(* CODESYS project SM_RTD.library
   Description: Device support for RTD Data Acquisition 8-Layer Stackable HAT for Raspberry Pi
   Version: 1.1.0.0
   Title: Raspberry I2C RTD Data Acquisition
   Author: Sequent Microsystems
   DocFormat: reStructuredText
   Placeholder: PlaceholderTemplate
   LanguageModelAttribute: qualified-access-only
   Company: Sequent Microsystems
   DefaultNamespace: SM_RTD

Project tree, tasks and I/O mapping:
  libraries: Raspberry Pi Peripherals, 4.6.0.0 (3S - Smart Software Solutions GmbH); IoStandard, 3.5.17.0 (System); Standard, 3.5.18.0 (System)
  global variables GVL
  function block SM_RTD [ST]: AfterReadInputs, BeforeWriteOutputs
  Library Information/
    function GetLibVersionNumber [ST]
    function GetLibVersion [ST]
    function IsLibReleased [ST]
  Project Information/
    function GetCompany [ST]
    function GetTitle [ST]
    function GetVersion [ST]
    function GetTextProperty [ST]
    function GetTextProperty2 [ST]
    function GetNumberProperty [ST]
    function GetBooleanProperty [ST]
    function GetVersionProperty [ST]
  data type REAL_UNION
*)

// REAL_UNION
TYPE REAL_UNION :
UNION
	rVal: REAL;
	b : ARRAY[0..3] OF BYTE;
END_UNION
END_TYPE

// GVL
//{attribute 'qualified_only'}
VAR_GLOBAL CONSTANT
	RTD_VAL_ADD: USINT := 16#00;	
END_VAR

// SM_RTD
FUNCTION_BLOCK SM_RTD EXTENDS i2c
VAR_INPUT
	//relayState: ARRAY[0..7] OF BOOL;
END_VAR
VAR_OUTPUT
	inRtdTemp: ARRAY[0..7] OF REAL;
END_VAR
VAR
	timer: TON := (IN:=TRUE);
END_VAR
VAR_TEMP	
	i, usi: USINT;
	buff: ARRAY[0..20] OF USINT;	
END_VAR

SUPER^();

CASE _iState OF
0:
	IF usiAddress < 16#40 OR  usiAddress > 16#47 THEN
		usiAddress := 16#40;
	END_IF
	
	IF SUPER^.init() THEN
		_iState := 5;
	END_IF	
5:	
	Timer.pt := T#25MS;
	
	// no initialisation here
	
	
	_iState := 10;
END_CASE

METHOD AfterReadInputs:INT
VAR
	Buffer : ARRAY[0..3] OF BYTE;
	ch: USINT;
	address: USINT;
	value: REAL_UNION;
	len: DINT;	
END_VAR
SUPER^.AfterReadInputs();

IF _iState = 10 THEN
	timer(IN:=TRUE);
	IF timer.Q THEN	
		FOR ch:=0 TO 7 DO
			address:= RTD_VAL_ADD + 4*ch;
			len := readregister(address, ADR(Buffer), 4);		
			IF len = 4 THEN
				value.b := Buffer;
				inRtdTemp[ch] := value.rVal;
				
			END_IF
		END_FOR
		
		timer(IN:=FALSE);
	END_IF
END_IF
END_METHOD

METHOD BeforeWriteOutputs:INT
VAR
	i: USINT;
	cnt: USINT;
	inVal:UINT;
	inSVal:USINT;
	buff: ARRAY[0..2] OF USINT;
	wStat: BOOL;
END_VAR
SUPER^.BeforeWriteOutputs();

IF _iState = 10 THEN

//nothing to write			
END_IF
END_METHOD

END_FUNCTION_BLOCK

// Library Information/GetLibVersionNumber
// This function has been automatically generated from the project information.
FUNCTION GetLibVersionNumber : DWORD
VAR_INPUT
	
END_VAR

GetLibVersionNumber := 16842752;

END_FUNCTION

// Project Information/GetCompany
// This function has been automatically generated from the project information.
{attribute 'signature_flag' := '1073741824'}
{attribute 'register_in_runtime'}
FUNCTION GetCompany : WSTRING
VAR_INPUT
	
END_VAR

GetCompany := "Sequent Microsystems";

END_FUNCTION

// Project Information/GetTitle
// This function has been automatically generated from the project information.
{attribute 'signature_flag' := '1073741824'}
{attribute 'register_in_runtime'}
FUNCTION GetTitle : WSTRING
VAR_INPUT
	
END_VAR

GetTitle := "Raspberry I2C RTD Data Acquisition";

END_FUNCTION

// Library Information/GetLibVersion
// This function has been automatically generated from the project information.
FUNCTION GetLibVersion : VERSION
VAR_INPUT
	
END_VAR

GetLibVersion.uiMajor := 1;
GetLibVersion.uiMinor := 1;
GetLibVersion.uiServicePack := 0;
GetLibVersion.uiPatch := 0;

END_FUNCTION

// Library Information/IsLibReleased
// This function has been automatically generated from the project information.
FUNCTION IsLibReleased : BOOL
VAR_INPUT
	
END_VAR

IsLibReleased := FALSE;

END_FUNCTION

// Project Information/GetVersion
// This function has been automatically generated from the project information.
{attribute 'signature_flag' := '1073741824'}
{attribute 'register_in_runtime'}
FUNCTION GetVersion : VERSION
VAR_INPUT
	
END_VAR

GetVersion.uiMajor := 1;
GetVersion.uiMinor := 1;
GetVersion.uiServicePack := 0;
GetVersion.uiPatch := 0;

END_FUNCTION

// Project Information/GetTextProperty
// This function has been automatically generated from the project information.
{attribute 'signature_flag' := '1073741824'}
{attribute 'register_in_runtime'}
FUNCTION GetTextProperty : WSTRING
VAR_INPUT
	stKey: WSTRING;
END_VAR

IF stKey = "Author" THEN
	GetTextProperty := "Sequent Microsystems";
ELSIF stKey = "Company" THEN
	GetTextProperty := "Sequent Microsystems";
ELSIF stKey = "DefaultNamespace" THEN
	GetTextProperty := "SM_RTD";
ELSIF stKey = "Description" THEN
	GetTextProperty := "Device support for RTD Data Acquisition 8-Layer Stackable HAT for Raspberry Pi";
ELSIF stKey = "DocFormat" THEN
	GetTextProperty := "reStructuredText";
ELSIF stKey = "LanguageModelAttribute" THEN
	GetTextProperty := "qualified-access-only";
ELSIF stKey = "Placeholder" THEN
	GetTextProperty := "PlaceholderTemplate";
ELSIF stKey = "Project" THEN
	GetTextProperty := "SM_RTD";
ELSIF stKey = "Title" THEN
	GetTextProperty := "Raspberry I2C RTD Data Acquisition";
ELSE
	GetTextProperty := "";
END_IF

END_FUNCTION

// Project Information/GetTextProperty2
// This function has been automatically generated from the project information.
{attribute 'signature_flag' := '1073741824'}
{attribute 'register_in_runtime'}
FUNCTION GetTextProperty2 : POINTER TO WSTRING
VAR_INPUT
	stKey: WSTRING;
END_VAR

IF stKey = "Author" THEN
	GetTextProperty2 := ADR("Sequent Microsystems");
ELSIF stKey = "Company" THEN
	GetTextProperty2 := ADR("Sequent Microsystems");
ELSIF stKey = "DefaultNamespace" THEN
	GetTextProperty2 := ADR("SM_RTD");
ELSIF stKey = "Description" THEN
	GetTextProperty2 := ADR("Device support for RTD Data Acquisition 8-Layer Stackable HAT for Raspberry Pi");
ELSIF stKey = "DocFormat" THEN
	GetTextProperty2 := ADR("reStructuredText");
ELSIF stKey = "LanguageModelAttribute" THEN
	GetTextProperty2 := ADR("qualified-access-only");
ELSIF stKey = "Placeholder" THEN
	GetTextProperty2 := ADR("PlaceholderTemplate");
ELSIF stKey = "Project" THEN
	GetTextProperty2 := ADR("SM_RTD");
ELSIF stKey = "Title" THEN
	GetTextProperty2 := ADR("Raspberry I2C RTD Data Acquisition");
ELSE
	GetTextProperty2 := ADR("");
END_IF

END_FUNCTION

// Project Information/GetNumberProperty
// This function has been automatically generated from the project information.
{attribute 'signature_flag' := '1073741824'}
{attribute 'register_in_runtime'}
FUNCTION GetNumberProperty : DINT
VAR_INPUT
	stKey: WSTRING;
END_VAR

GetNumberProperty := 0;

END_FUNCTION

// Project Information/GetBooleanProperty
// This function has been automatically generated from the project information.
{attribute 'signature_flag' := '1073741824'}
{attribute 'register_in_runtime'}
FUNCTION GetBooleanProperty : BOOL
VAR_INPUT
	stKey: WSTRING;
END_VAR

IF stKey = "IsEndUserLibrary" THEN
	GetBooleanProperty := FALSE;
ELSIF stKey = "Released" THEN
	GetBooleanProperty := FALSE;
ELSE
	GetBooleanProperty := FALSE;
END_IF

END_FUNCTION

// Project Information/GetVersionProperty
// This function has been automatically generated from the project information.
{attribute 'signature_flag' := '1073741824'}
{attribute 'register_in_runtime'}
FUNCTION GetVersionProperty : VERSION
VAR_INPUT
	stKey: WSTRING;
END_VAR

IF stKey = "Version" THEN
	GetVersionProperty.uiMajor := 1;
	GetVersionProperty.uiMinor := 1;
	GetVersionProperty.uiServicePack := 0;
	GetVersionProperty.uiPatch := 0;
ELSE
	GetVersionProperty.uiMajor := 0;
	GetVersionProperty.uiMinor := 0;
	GetVersionProperty.uiServicePack := 0;
	GetVersionProperty.uiPatch := 0;
END_IF

END_FUNCTION
